// TIA Portal V17 export
// export: Created 2024-08-09T12:53:24.1948839Z, ExportSetting WithDefaults, DisplayName Totally Integrated Automation Portal, DisplayVersion V17 Update 7, DisplayName TIA Portal Openness, DisplayVersion V17 Update 7, DisplayName TIA Portal Version Control Interface, DisplayVersion V17, DisplayName STEP 7 Professional, DisplayVersion V17 Update 7, DisplayName STEP 7 Safety, DisplayVersion V17 Update 6, DisplayName WinCC Professional, DisplayVersion V17 Update 7
TYPE "Case"
// stored: IsFailsafeCompliant false
   STRUCT
      Matiere : String[20];
      Zone : String[16];
      Code_Couleur : String;
      T_Remplissage : Real;
      Quantite : Real;
      Volume : Real;
      Densite : Real;
   END_STRUCT;
END_TYPE
